// TIA Portal project "HMI_Cl2_Liquid_Tanks_New" (V20)

(* hardware
DEVICE "S7-1500/ET200MP station_1"  S7-1500 station
   slot 0: "Rail_0"  Rack  6ES7 590-1***0-0AA0
   slot 1: "PLC_1"  CPU 1511-1 PN  6ES7 511-1AK02-0AB0  V2.9
      slot 3: "CPU display_1"  6ES7591-1AA00-0AA0
      slot 32768: "PROFINET interface_1"  X1
         slot 32769: "Port_1"  X1 P1
         slot 32770: "Port_2"  X1 P2
      slot 34817: "Virtual CP interface port_1"  Virtual CP interface port  Virtual CP interface port
DEVICE "PC-System_1"  SIMATIC PC station
   slot 0: "SIMATIC PC station"  Rail  SIMATIC PC-Station  V1.0
      slot 125: "Stationmanager"  Station_Manager  V6.0.4
   slot 1: "HMI_RT_1"  WinCC RT Advanced  6AV2 104-0xxxx-xxxx  17.0.0.0
      slot 33792: "Computer interface"  Host interface
   slot 2: "IE general_1"  IE General  IE_CP  V8.2.0
      slot 1: "PROFINET interface"  IEGeneral.Interface.8.2.0
*)

// ===== PLC "PLC_1"  CPU 1511-1 PN =====

DATA_BLOCK "DB_HMI_Cl2"   // DB1
{ S7_Optimized_Access := 'TRUE' }
VERSION : 0.1
   VAR
      TankTemp_C : Real;
      TempSensorFault : Bool;
      AutoModeActive : Bool;
      AlarmActive : Bool;
      AlarmBits : Int;
   END_VAR
BEGIN
END_DATA_BLOCK

DATA_BLOCK "FB_Cl2Demo_DB"   // DB2
{ S7_Optimized_Access := 'TRUE' }
VERSION : 0.1
// stored: InstanceOfName FB_Cl2Demo
"FB_Cl2Demo"
BEGIN
END_DATA_BLOCK

FUNCTION_BLOCK "FB_Cl2Demo"   // FB1, SCL
{ S7_Optimized_Access := 'TRUE' }
// PLC_1 / TIA Portal V20 / S7-PLCSIM ONLY.
//  One call per SECOND in a cyclic interrupt OB. No physical I/O is read/written.
//  Illustrative values are not operating setpoints or protective limits.
//  Write ONLY these commands from HMI or a PLCSIM watch table.
   VAR
      SimEnable : Bool := FALSE;
      RunRequest : Bool := FALSE;
      AutoModeRequest : Bool := FALSE;   // Display only; no automatic control logic.
      InjectTempFault : Bool := FALSE;
      InjectCoolingFault : Bool := FALSE;
      InjectAcidFault : Bool := FALSE;
      InjectK805Fault : Bool := FALSE;
      DemoCoolingAlarmWord : Word := WORD#16#0000;   // Read-only process indication for HMI. Do not set these from HMI.
      Stage : Int := 0;   // 0 stopped; 1 E801; 2 drying; 3 K805; 4 separators; 5 E809; 6 storage.
      Tick : DInt := 0;   // In seconds IF called from 1 s OB.
      E801Running : Bool := FALSE;
      DryersRunning : Bool := FALSE;
      K805Running : Bool := FALSE;
      D805Running : Bool := FALSE;
      F805Running : Bool := FALSE;
      CoolingRunning : Bool := FALSE;
      E809Running : Bool := FALSE;
      TankFillActive : Bool := FALSE;
      AutoModeActive : Bool := FALSE;
      TempSensorFault : Bool := FALSE;
      CoolingFault : Bool := FALSE;
      AcidFault : Bool := FALSE;
      K805Fault : Bool := FALSE;
      AlarmActive : Bool := FALSE;
      ProcessHealthy : Bool := FALSE;   // Demo measurements (units are in names; independent of real I/O).
      TankTemp_C : Real := 25.5;
      E801_GasOut_C : Real := 23.5;
      C804_Acid_C : Real := 18.5;
      C805_Acid_C : Real := 18.5;
      C804_Acid_pct : Real := 80.0;
      C805_Acid_pct : Real := 90.0;
      K805_Acid_pct : Real := 98.0;
      K805_GasIn_C : Real := 29.0;
      D805_P_kgcm2 : Real := 0.0;
      E809_P_kgcm2 : Real := 0.0;
      E809_Temp_C : Real := 23.5;
      D807_R22_P_kgcm2 : Real := 0.0;
      D822_Level_pct : Real := 10.0;
      D823_Level_pct : Real := 10.0;
      D824_Level_pct : Real := 10.0;
      D825_Level_pct : Real := 10.0;   // Internal edge state; not connected to the HMI.
      LastSimEnable : Bool := FALSE;
   END_VAR
BEGIN

   // An explicit enable separates this training model from a real PLC program.
   IF NOT #SimEnable THEN
       #Stage := 0;
       #Tick := 0;
       #E801Running := FALSE;
       #DryersRunning := FALSE;
       #K805Running := FALSE;
       #D805Running := FALSE;
       #F805Running := FALSE;
       #CoolingRunning := FALSE;
       #E809Running := FALSE;
       #TankFillActive := FALSE;
       #AutoModeActive := FALSE;
       #TempSensorFault := FALSE;
       #CoolingFault := FALSE;
       #AcidFault := FALSE;
       #K805Fault := FALSE;
       #AlarmActive := FALSE;
       #ProcessHealthy := FALSE;
       #D805_P_kgcm2 := 0.0;
       #E809_P_kgcm2 := 0.0;
       #D807_R22_P_kgcm2 := 0.0;
       #LastSimEnable := FALSE;
       #DemoCoolingAlarmWord := W#16#0000;
       RETURN;
   END_IF;

   // Reset synthetic measurements at the beginning of a new demo session.
   IF NOT #LastSimEnable THEN
       #TankTemp_C := 25.5;
       #E801_GasOut_C := 23.5;
       #C804_Acid_C := 18.5;
       #C805_Acid_C := 18.5;
       #C804_Acid_pct := 80.0;
       #C805_Acid_pct := 90.0;
       #K805_Acid_pct := 98.0;
       #K805_GasIn_C := 29.0;
       #E809_Temp_C := 23.5;
       #D822_Level_pct := 10.0;
       #D823_Level_pct := 10.0;
       #D824_Level_pct := 10.0;
       #D825_Level_pct := 10.0;
       #Tick := 0;
   END_IF;
   #LastSimEnable := TRUE;

   #AutoModeActive := #AutoModeRequest;
   #TempSensorFault := #InjectTempFault;
   #CoolingFault := #InjectCoolingFault;
   #DemoCoolingAlarmWord.%X0 := #CoolingFault;
   #AcidFault := #InjectAcidFault;
   #K805Fault := #InjectK805Fault;
   #AlarmActive := #TempSensorFault OR #CoolingFault OR #AcidFault OR #K805Fault;

   IF #AcidFault THEN
       // Deliberately off-normal SAMPLE values; these are not trip settings.
       #C804_Acid_pct := 70.0;
       #C805_Acid_pct := 80.0;
       #K805_Acid_pct := 93.0;
   ELSE
       #C804_Acid_pct := 80.0;
       #C805_Acid_pct := 90.0;
       #K805_Acid_pct := 98.0;
   END_IF;

   IF #RunRequest THEN
       IF #Tick < 3600 THEN
           #Tick := #Tick + 1;
       END_IF;
       IF #Tick < 2 THEN
           #Stage := 0;
       ELSIF #Tick < 4 THEN
           #Stage := 1;
       ELSIF #Tick < 6 THEN
           #Stage := 2;
       ELSIF #Tick < 8 THEN
           #Stage := 3;
       ELSIF #Tick < 10 THEN
           #Stage := 4;
       ELSIF #Tick < 12 THEN
           #Stage := 5;
       ELSE
           #Stage := 6;
       END_IF;
   ELSE
       #Tick := 0;
       #Stage := 0;
   END_IF;

   #E801Running := #Stage >= 1;
   #DryersRunning := #Stage >= 2;
   #K805Running := (#Stage >= 3) AND NOT #K805Fault;
   #D805Running := (#Stage >= 4) AND #K805Running;
   #F805Running := #D805Running;
   #CoolingRunning := (#Stage >= 5) AND NOT #CoolingFault;
   #E809Running := (#Stage >= 5) AND #F805Running AND #CoolingRunning;
   #TankFillActive := (#Stage >= 6) AND #E809Running AND NOT #AcidFault;
   #ProcessHealthy := (#Stage >= 6) AND NOT #AlarmActive;

   // Approximate values for a visual simulation, NOT a thermodynamic model.
   IF #K805Running THEN
       #D805_P_kgcm2 := 2.5;
   ELSE
       #D805_P_kgcm2 := 0.0;
   END_IF;
   IF #CoolingRunning THEN
       #D807_R22_P_kgcm2 := 12.0;
   ELSE
       #D807_R22_P_kgcm2 := 0.0;
   END_IF;
   IF #E809Running THEN
       #E809_P_kgcm2 := 1.0;
       IF #E809_Temp_C > -15.0 THEN
           #E809_Temp_C := #E809_Temp_C - 0.5;
           IF #E809_Temp_C < -15.0 THEN
               #E809_Temp_C := -15.0;
           END_IF;
       END_IF;
   ELSE
       #E809_P_kgcm2 := 0.0;
       IF #E809_Temp_C < 23.5 THEN
           #E809_Temp_C := #E809_Temp_C + 0.4;
           IF #E809_Temp_C > 23.5 THEN
               #E809_Temp_C := 23.5;
           END_IF;
       END_IF;
   END_IF;

   // Time-compressed tank animation, not a material balance calculation.
   IF #TankFillActive AND ((#Tick MOD 5) = 0) THEN
       IF #D822_Level_pct < 80.0 THEN
           #D822_Level_pct := #D822_Level_pct + 1.0;
       ELSIF #D823_Level_pct < 80.0 THEN
           #D823_Level_pct := #D823_Level_pct + 1.0;
       ELSIF #D824_Level_pct < 80.0 THEN
           #D824_Level_pct := #D824_Level_pct + 1.0;
       ELSIF #D825_Level_pct < 80.0 THEN
           #D825_Level_pct := #D825_Level_pct + 1.0;
       END_IF;
   END_IF;
END_FUNCTION_BLOCK

FUNCTION "FC_AlarmDemo" : Void   // FC1, SCL
{ S7_Optimized_Access := 'TRUE' }
VERSION : 0.1
BEGIN
   "DB_HMI_Cl2".AlarmActive := "DB_HMI_Cl2".TempSensorFault;
   "DB_HMI_Cl2".AlarmBits := BOOL_TO_INT("DB_HMI_Cl2".TempSensorFault);
END_FUNCTION

ORGANIZATION_BLOCK "Main"   // OB1, LAD, ProgramCycle
TITLE = "Main Program Sweep (Cycle)"
{ S7_Optimized_Access := 'TRUE' }
VERSION : 0.1
   VAR_INPUT
      Initial_Call : Bool;   // Initial call of this OB
      Remanence : Bool;   // =True, if remanent data are available
   END_VAR
BEGIN

REGION Network 1
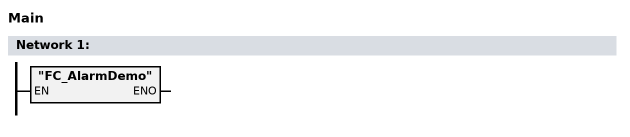
   RUNG wire#powerrail
      "FC_AlarmDemo"()
   END_RUNG
   // the same network as SCL:
   "FC_AlarmDemo"();
END_REGION
END_ORGANIZATION_BLOCK

ORGANIZATION_BLOCK "CyclicInterrupt"   // OB30, LAD, CyclicInterrupt
{ S7_Optimized_Access := 'TRUE' }
VERSION : 0.1
   VAR_INPUT
      Initial_Call : Bool;   // Initial call of this OB
      Event_Count : Int;   // Events discarded
   END_VAR
BEGIN

REGION Network 1
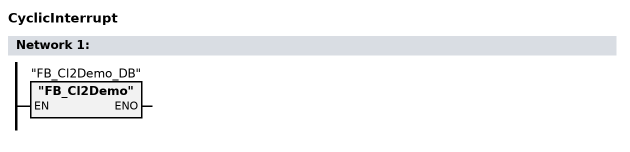
   RUNG wire#powerrail
      "FB_Cl2Demo_DB"()
   END_RUNG
   // the same network as SCL:
   "FB_Cl2Demo_DB"();   // "FB_Cl2Demo"
END_REGION
END_ORGANIZATION_BLOCK

(* ===== HMI "HMI_RT_1" =====
system functions are stored by id; their names below are inferred from use
connection "HMI_Connection_1": ETHERNET, S7_1500_OMS

HMI tags "Default tag table"
   "TankTemp_C" : Real = PLC DB_HMI_Cl2.TankTemp_C AT %DB1.DBW0, 1 s
   "TempSensorFault" : Bool = PLC DB_HMI_Cl2.TempSensorFault AT %DB1.DBD0, 1 s
   "AutoModeActive" : Bool = PLC DB_HMI_Cl2.AutoModeActive AT %DB1.DBX0.0, 1 s
   "AlarmActive" : Bool = PLC DB_HMI_Cl2.AlarmActive AT %DB1.DBX0.0, 1 s
   "AlarmBits" : Int = PLC DB_HMI_Cl2.AlarmBits AT %DB1.DBW0, 1 s
   "DemoStage" : Int = PLC FB_Cl2Demo_DB.Stage AT %DB1.DBW0, 1 s
   "DemoE809Temp" : Real = PLC FB_Cl2Demo_DB.E809_Temp_C AT %DB1.DBD0, 1 s
   "DemoE801Running" : Bool = PLC FB_Cl2Demo_DB.E801Running AT %DB1.DBX0.0, 1 s
   "DemoK805Running" : Bool = PLC FB_Cl2Demo_DB.K805Running AT %DB1.DBX0.0, 1 s
   "DemoD822Level" : Real = PLC FB_Cl2Demo_DB.D822_Level_pct AT %DB1.DBX0.0, 1 s
   "DemoRunRequest" : Bool = PLC FB_Cl2Demo_DB.RunRequest AT %DB1.DBD0, 1 s
   "DemoInjectK805Fault" : Bool = PLC FB_Cl2Demo_DB.InjectK805Fault AT %DB1.DBX0.0, 1 s
   "DemoDryersRunning" : Bool = PLC FB_Cl2Demo_DB.DryersRunning AT %DB1.DBX0.0, 1 s
   "DemoD805Running" : Bool = PLC FB_Cl2Demo_DB.D805Running AT %DB1.DBX0.0, 1 s
   "DemoF805Running" : Bool = PLC FB_Cl2Demo_DB.F805Running AT %DB1.DBX0.0, 1 s
   "DemoCoolingRunning" : Bool = PLC FB_Cl2Demo_DB.CoolingRunning AT %DB1.DBX0.0, 1 s
   "DemoE809Running" : Bool = PLC FB_Cl2Demo_DB.E809Running AT %DB1.DBX0.0, 1 s
   "DemoTankFillActive" : Bool = PLC FB_Cl2Demo_DB.TankFillActive AT %DB1.DBX0.0, 1 s
   "DemoD824Level" : Real = PLC FB_Cl2Demo_DB.D824_Level_pct AT %DB1.DBX0.0, 1 s
   "DemoD825Level" : Real = PLC FB_Cl2Demo_DB.D825_Level_pct AT %DB1.DBD0, 1 s
   "DemoE809Pressure" : Real = PLC FB_Cl2Demo_DB.E809_P_kgcm2 AT %DB1.DBD0, 1 s
   "DemoR22Pressure" : Real = PLC FB_Cl2Demo_DB.D807_R22_P_kgcm2 AT %DB1.DBD0, 1 s
   "DemoD823Level" : Real = PLC FB_Cl2Demo_DB.D823_Level_pct AT %DB1.DBX0.0, 1 s
   "DemoSimEnable" : Bool = PLC FB_Cl2Demo_DB.SimEnable AT %DB1.DBD0, 1 s
   "DemoCoolingAlarmWord" : Word = PLC FB_Cl2Demo_DB.DemoCoolingAlarmWord AT %DB1.DBW0, 1 s

discrete alarms
   1: 'LỖI CẢM BIẾN NHIỆT – không sử dụng giá trị nhiệt độ; kiểm tra cảm biến', class Errors, trigger "AlarmBits" bit 0
   2: '“Lỗi làm lạnh R22 – kiểm tra mạch lạnh và E809', class Errors, trigger "DemoCoolingAlarmWord" bit 0

screen "Overview_Cl2" 1024x768
   TextField "Text field_1" at 347,14 size 218x22; Text 'BỂ CLO LỎNG – TỔNG QUAN'
   IOField "I/O field_1" at 141,255 size 96x32; FormatPattern 999.9
      ProcessValue <- "TankTemp_C"
      Visibility <- "TempSensorFault"
   TextField "Text field_2" at 9,254 size 95x22; Text 'Nhiệt độ bể:'
   TextField "Text field_3" at 313,254 size 168x22; Text 'LỖI CẢM BIẾN NHIỆT'
      Visibility <- "AlarmActive"
   TextField "Text field_4" at 141,255 size 154x22; Text 'KHÔNG CÓ DỮ LIỆU'
      Visibility <- "TempSensorFault"
   TextField "Text field_5" at 841,13 size 60x22; Text 'Chế độ:'
   TextField "Text field_6" at 913,12 size 77x22; Text 'TỰ ĐỘNG'
      Visibility <- "AutoModeActive"
   TextField "Text field_7" at 906,14 size 85x22; Text 'THỦ CÔNG'
      Visibility <- "AutoModeActive"
   TrendView "Trend view_1" at 0,507 size 540x261
   IOField "I/O field_2" at 140,92 size 96x32; FormatPattern 9
      ProcessValue <- "DemoStage"
   TextField "Text field_8" at 9,95 size 80x22; Text 'Giai đoạn:'
   TextField "Text field_9" at 12,150 size 116x22; Text 'Nhiệt độ E809:'
   IOField "I/O field_3" at 141,147 size 96x32; FormatPattern 999.9
      ProcessValue <- "DemoE809Temp"
   Circle "Circle_1" at 249,150 size 24x24
      Appearance <- "DemoE801Running"
   TextField "Text field_10" at 10,203 size 130x22; Text 'Trạng thái K805:'
   Circle "Circle_2" at 171,199 size 37x37
      Appearance <- "DemoK805Running"
   Bar "Bar_1" at 606,544 size 74x215; MinimumValue 0; MaximumValue 100
      ProcessValue <- "DemoD822Level"
   TextField "Text field_11" at 622,518 size 46x22; Text 'D822'
   Button "Button_1" at 10,46 size 96x32; TextOff 'Run'
      on Click: SetBit("DemoRunRequest")
      Appearance <- "DemoRunRequest"
   Button "Button_2" at 129,46 size 96x32; TextOff 'Stop'
      on Click: ResetBit("DemoRunRequest")
      Appearance <- "DemoRunRequest"
   Bar "Bar_2" at 802,544 size 74x215; MinimumValue 0; MaximumValue 100
      ProcessValue <- "DemoD824Level"
   GraphicView "Graphic view_3" at 295,38 size 100x100; Picture "E809_hoa_long"
   GraphicView "Graphic view_1" at 396,36 size 100x100; Picture "C804_thap_say"
   GraphicView "Graphic view_4" at 444,40 size 100x100; Picture "rfo2irvv.q3j"
   GraphicView "Graphic view_2" at 898,32 size 100x100; Picture "Bon_Clo_long"
   GraphicView "Graphic view_5" at 539,36 size 100x100; Picture "K805_may_nen_clo"
   GraphicView "Graphic view_6" at 631,38 size 100x100; Picture "D805_tach_long"
   GraphicView "Graphic view_9" at 628,172 size 100x100; Picture "K805_may_nen_clo"
   GraphicView "Graphic view_10" at 750,172 size 100x100; Picture "E809_hoa_long"
   GraphicView "Graphic view_11" at 833,168 size 100x100; Picture "D807_binh_chua_R22"
   GraphicView "Graphic view_12" at 924,172 size 100x100; Picture "E808_bay_hoi"
   GraphicView "Graphic view_14" at 697,40 size 100x100; Picture "F805_tach_mu"
   GraphicView "Graphic view_17" at 781,32 size 100x100; Picture "tfat2e1y.sgp"
   Line "Line_1" at 385,89 size 48x1
      Visibility <- "DemoDryersRunning"
   Line "Line_2" at 506,90 size 37x1
      Visibility <- "DemoK805Running"
   Line "Line_4" at 633,88 size 32x1
      Visibility <- "DemoD805Running"
   Line "Line_5" at 704,76 size 31x1
      Visibility <- "DemoF805Running"
   Line "Line_6" at 756,84 size 29x0
      Visibility <- "DemoE809Running"
   Line "Line_7" at 876,82 size 33x0
      Visibility <- "DemoTankFillActive"
   Line "Line_8" at 720,222 size 34x1
      Visibility <- "DemoCoolingRunning"
   Line "Line_9" at 845,220 size 30x1
      Visibility <- "DemoCoolingRunning"
   Line "Line_10" at 891,219 size 42x2
      Visibility <- "DemoCoolingRunning"
   Line "Line_11" at 969,125 size 0x85
      Visibility <- "DemoCoolingRunning"
   Line "Line_12" at 857,128 size 114x4
      Visibility <- "DemoCoolingRunning"
   Line "Line_13" at 862,94 size 1x38
      Visibility <- "DemoCoolingRunning"
   Line "Line_14" at 790,95 size 0x48
      Visibility <- "DemoCoolingRunning"
   Line "Line_16" at 684,142 size 106x1
      Visibility <- "DemoCoolingRunning"
   Line "Line_17" at 686,144 size 0x72
      Visibility <- "DemoCoolingRunning"
   TextField "Text field_12" at 327,119 size 44x22; Text 'E801'
   TextField "Text field_13" at 428,132 size 94x22; Text 'C804/C805'
   TextField "Text field_14" at 573,121 size 45x22; Text 'K805'
   TextField "Text field_15" at 661,125 size 46x22; Text 'D805'
   TextField "Text field_16" at 732,121 size 44x22; Text 'F805'
   TextField "Text field_17" at 805,105 size 44x22; Text 'E809'
   TextField "Text field_18" at 892,105 size 101x22; Text 'Bồn Clo Lỏng'
   TextField "Text field_19" at 955,236 size 44x22; Text 'E808'
   TextField "Text field_20" at 863,248 size 46x22; Text 'D807'
   TextField "Text field_21" at 781,246 size 44x22; Text 'E807'
   TextField "Text field_22" at 661,248 size 56x22; Text 'KR801'
   TextField "Text field_23" at 236,62 size 61x22; Text 'Khí CLo'
   Line "Line_3" at 276,90 size 24x0
      Visibility <- "DemoE801Running"
   Bar "Bar_3" at 906,544 size 74x215; MinimumValue 0; MaximumValue 100
      ProcessValue <- "DemoD825Level"
   TextField "Text field_24" at 814,519 size 46x22; Text 'D824'
   TextField "Text field_25" at 918,519 size 46x22; Text 'D825'
   IOField "I/O field_4" at 792,138 size 96x32; FormatPattern 999.99
      ProcessValue <- "DemoE809Pressure"
   IOField "I/O field_5" at 844,268 size 96x32; FormatPattern 999.99
      ProcessValue <- "DemoR22Pressure"
   Bar "Bar_4" at 703,544 size 74x215; MinimumValue 0; MaximumValue 100
      ProcessValue <- "DemoD823Level"
   TextField "Text field_26" at 713,518 size 46x22; Text 'D823'
   Button "Button_3" at 141,451 size 96x32; TextOff 'Start'
      on Click: SetBit("DemoSimEnable")
      Appearance <- "DemoSimEnable"
   Button "Button_4" at 251,450 size 96x32; TextOff 'End'
      on Activate: ResetBit("DemoSimEnable")
      Appearance <- "DemoSimEnable"
   TextField "Text field_27" at 5,451 size 122x22; Text 'Chạy mô phỏng:'
   Button "Button_5" at 432,451 size 96x32; TextOff 'Cảnh báo'
      on Click: ActivateScreen("Alarms_Cl2", 0)
   TextField "Text field_28" at 15,304 size 112x22; Text 'Áp suất E809:'
   IOField "I/O field_6" at 141,300 size 96x32; FormatPattern 999.99
      ProcessValue <- "DemoE809Pressure"
   TextField "Text field_29" at 19,358 size 100x22; Text 'Áp suất R22:'
   IOField "I/O field_7" at 140,356 size 96x32; FormatPattern 999.99
      ProcessValue <- "DemoR22Pressure"
   Circle "Circle_3" at 618,106 size 26x26
      Appearance <- "DemoK805Running"
   Circle "Circle_4" at 867,95 size 22x22
      Appearance <- "DemoE809Running"
   Circle "Circle_5" at 727,236 size 24x24
      Appearance <- "DemoCoolingRunning"
   Button "Button_6" at 722,387 size 195x82; TextOff 'Dừng khẩn cấp'
   Circle "Circle_6" at 371,118 size 15x15
      Appearance <- "DemoE801Running"
   Circle "Circle_7" at 519,118 size 14x14
      Appearance <- "DemoDryersRunning"
   Circle "Circle_8" at 699,119 size 14x14
      Appearance <- "DemoD805Running"
   Circle "Circle_9" at 767,109 size 14x14
      Appearance <- "DemoF805Running"
   TextField "Text field_30" at 759,303 size 115x22; Text 'Mạch lạnh R22'

screen "Alarms_Cl2" 1024x768
   AlarmView "Alarm view_1" at 199,78 size 600x300
   Button "Button_1" at 7,18 size 192x32; TextOff 'Quay Lại'; TextOn 'Overview_Cl2'
      on Click: ActivateScreen("Overview_Cl2", 0)
*)